(* IEC 61131-3 sources: ATCMcontrol_Engineering/src/TargetBase/Libs/MectUserUtility, 8 files *)

(* ---- Buzzer.st ---- *)
(*[[
    UserHelpURL= "ATCMfile:Buzzer.HTML",
]]*)
FUNCTION Buzzer : UINT
VAR_INPUT
	duration : UINT; (*[duration in ms]*)
END_VAR
	INLINE {STDLIB(Buzzer)}
END_FUNCTION

(* ---- Date_add.st ---- *)
(*[[
    UserHelpURL= "ATCMfile:Date_add.HTML",
]]*)
FUNCTION Date_add : STRING
VAR_INPUT
	initDate  : STRING; (*[ starting date in format "DD-MM-YYYY" ]*)
	format    : STRING; (*[ "D" for days, "W" for weeks, "M" for months and "Y" for years ]*)
	increment : INT; (*[ value to add ]*)
END_VAR
VAR_OUTPUT
	finalDate     : STRING; (*[ starting date in format "DD-MM-YYYY" ]*)
END_VAR
	INLINE {STDLIB(Date_add)}
END_FUNCTION

(* ---- Date_diff.st ---- *)
(*[[
    UserHelpURL= "ATCMfile:Date_diff.HTML",
]]*)
FUNCTION Date_diff : UINT
VAR_INPUT
	initDate  : STRING; (*[ starting date in format "DD-MM-YYYY" ]*)
	finalDate : STRING; (*[ end date in format "DD-MM-YYYY" ]*)
	format    : STRING; (*[ "D" for days, "W" for weeks, "M" for months and "Y" for years ]*)
END_VAR
VAR_OUTPUT
	diff      : DINT; (*[ difference between start date and end date expressed in "format" ]*)
END_VAR
	INLINE {STDLIB(Date_diff)}
END_FUNCTION

(* ---- DateTimeRead.st ---- *)
(*[[
    UserHelpURL= "ATCMfile:DateTimeRead.HTML",
]]*)
FUNCTION DateTimeRead : UINT
VAR_OUTPUT
	DateTime : ARRAY[0..6] of UINT; (*[date in  YEAR, MONTH, DAY, HOUR, MINUTE, SECONDS]*)
END_VAR
	INLINE {STDLIB(DateTimeRead)}
END_FUNCTION

(* ---- DateTimeSync.st ---- *)
(*[[
    UserHelpURL= "ATCMfile:DateTimeSync.HTML",
]]*)
FUNCTION DateTimeSync : UINT
VAR_INPUT
END_VAR
	INLINE {STDLIB(DateTimeSync)}
END_FUNCTION

(* ---- DateTimeWrite.st ---- *)
(*[[
    UserHelpURL= "ATCMfile:DateTimeWrite.HTML",
]]*)
FUNCTION DateTimeWrite : UINT
VAR_INPUT
	DateTime : ARRAY[0..6] of UINT; (*[date in  YEAR, MONTH, DAY, HOUR, MINUTE, SECONDS]*)
END_VAR
	INLINE {STDLIB(DateTimeWrite)}
END_FUNCTION

(* ---- LCD_get_backlight.st ---- *)
(*[[
    UserHelpURL= "ATCMfile:LCD_get_backlight.HTML",
]]*)
FUNCTION LCD_get_backlight : UINT
VAR_OUTPUT
	DutyCycle : UINT; (*[ LCD PWM DutyCycle ]*)
END_VAR
	INLINE {STDLIB(LCD_get_backlight)}
END_FUNCTION

(* ---- LCD_set_backlight.st ---- *)
(*[[
    UserHelpURL= "ATCMfile:LCD_set_backlight.HTML",
]]*)
FUNCTION LCD_set_backlight : UINT
VAR_INPUT
	DutyCycle : UINT; (*[ LCD PWM DutyCycle ]*)
END_VAR
	INLINE {STDLIB(LCD_set_backlight)}
END_FUNCTION
